(* CODESYS project TCP Client Read Write Example.project

Project tree, tasks and I/O mapping:
  Device : CODESYS Control for Raspberry Pi, 3S - Smart Software Solutions GmbH, version 3.5.11.20
    application Application
      libraries: Standard, * (System); Network, 3.5.7.0 (3S - Smart Software Solutions GmbH); Raspberry I2C Gyroscopes, 1.1.1.0 (3S - Smart Software Solutions GmbH)
      task MainTask (cyclic, interval 4 ms, priority 1) calls PLC_PRG
      task VISU_TASK (cyclic, interval 100 ms, priority 31) calls VisuElems.Visu_Prg
      program PLC_PRG [CFC]
      visualisation Visualization
      function block TCP_Read_and_Write [ST]
    SoftMotion General Axis Pool
    I²C
    SPI
    GPIOs_A_B : GPIOs A/B, 3S - Smart Software Solutions GmbH, version 3.5.11.0
        unmapped channels: digital inputs (GPIO0..GPIO31), digital outputs (GPIO0..GPIO31)
    Onewire
    Camera device
      <Leer>
  text list GlobalTextList
*)

// Device/Application/PLC_PRG
PROGRAM PLC_PRG
VAR
	startRequest: BOOL;
	returnCode: INT;
	transmitData: STRING := 'Hello World!';
	done: BOOL;
	receiveData: STRING;
	clientConnection: TCP_Read_and_Write;
END_VAR

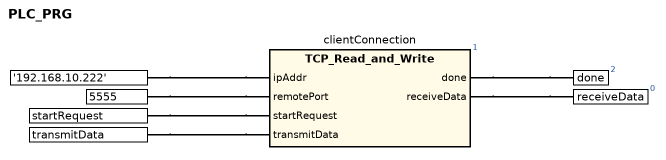
receiveData := clientConnection.receiveData;
clientConnection(
    ipAddr := '192.168.10.222',
    remotePort := 5555,
    startRequest := startRequest,
    transmitData := transmitData); // TCP_Read_and_Write
done := clientConnection.done;

END_PROGRAM

// Device/Application/TCP_Read_and_Write
FUNCTION_BLOCK TCP_Read_and_Write
VAR_INPUT
	ipAddr: STRING;
	remotePort: UINT;
	startRequest: BOOL;
	transmitData: STRING;
END_VAR
VAR_OUTPUT
	done: BOOL;
	receiveData: STRING;
END_VAR
VAR
	R_TRIG_StartRequest: R_TRIG;
	tcpClient: nbs.TCP_Client;
	tcpWrite: nbs.TCP_Write;
	tcpRead: nbs.TCP_Read;
    startSend : BOOL;
	targetAddr: NBS.IP_ADDR;
	iStep: INT := 0;
END_VAR


R_TRIG_StartRequest(CLK:=startRequest);
IF R_TRIG_StartRequest.Q THEN
	iStep := 10;
END_IF;

CASE iStep OF

	0: 

	10:
		// create connection to server
		done := FALSE;
		targetAddr.sAddr := ipAddr;
		tcpClient(xEnable:=TRUE, ipAddr:=targetAddr, uiPort:=remotePort);
		IF tcpClient.xActive THEN
			iStep := 20;  
		END_IF 
		
	20:
		// write string to opened connection
		tcpWrite(hConnection:=tcpClient.hConnection, xExecute:=TRUE, pData:=ADR(transmitData), szSize:=SIZEOF(transmitData));
		IF tcpWrite.xDone THEN
			tcpWrite(xExecute:=FALSE);
			iStep := 30;
		END_IF
		
	30:
		// wait for answer and read it
		tcpRead(hConnection:=tcpClient.hConnection, xEnable:=tcpClient.xActive, pData:=ADR(receiveData), szSize:=SIZEOF(receiveData));	
		IF tcpRead.xReady THEN
			iStep := 40;
		END_IF
		
	40:
		// close connection
		done := TRUE;
		tcpRead(xEnable:=FALSE);
		tcpClient(xEnable:=FALSE);
		iStep := 0;

END_CASE

END_FUNCTION_BLOCK

// Device/Application/Visualization
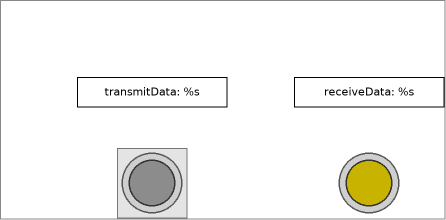
VISUALIZATION Visualization  // 446x220
    PushSwitch (117,148 70x70), variable: PLC_PRG.startRequest, behaviour: TAP, style: Switch-PushSwitch-Gray
    Rectangle (294,77 150x30), "receiveData: %s", text variable: PLC_PRG.receiveData
    Rectangle (77,77 150x30), "transmitData: %s", text variable: PLC_PRG.transmitData
    Lamp1 (334,148 70x70), variable: PLC_PRG.done, style: Lamp-Lamp1-Yellow
END_VISUALIZATION
